Fanuc KAREL source: kt00490.KL

-- PROVISIONAL review KL for V940-1; original PC SHA256 199719eee872a66ce0fa5f90e25866bc2ee3d830b8123261f9883592636b3d4f
-- Incomplete behavior may be omitted. Consult companion uncertainty JSON. Do not deploy.
PROGRAM KT00490
%NOLOCKGROUP
-- UNRESOLVED_DECL P1 type=000101
-- UNRESOLVED_DECL P2 type=000199
-- UNRESOLVED_DECL OUT type=000102
BEGIN
  -- V9_ZERO_TABLE_METADATA_HINT layout=0001; no indexed target words; source/name/runtime held
  -- UNRESOLVED_PC offsets 5-39; opcodes 49,49,7E,60,7E,4A
  -- UNRESOLVED_PC offsets 44-48; opcodes 7F
END KT00490
